(* IEC 61131-3 sources: Word/plc-course/07-timers/labs/starter, 5 files *)

(* ---- 07-1-star-delta.st ---- *)
(* Lab 07-1: Star-delta starter.
   Module 07 (Timers). STARTER - the declarations are done for you;
   write the logic where it says TODO, then run:
     python3 tools/plctest.py 07-timers/labs/starter/07-1-star-delta.st *)

PROGRAM StarDelta
  VAR (* I/O *)
    StartPB       AT %IX0.0 : BOOL;  (* Start push-button, NO: TRUE while pressed *)
    StopPB_NC     AT %IX0.1 : BOOL;  (* Stop push-button, NC: TRUE while NOT pressed *)
    OverloadOK_NC AT %IX0.2 : BOOL;  (* Overload relay contact, NC: TRUE while healthy *)
    MainK         AT %QX0.0 : BOOL;  (* Main (line) contactor *)
    StarK         AT %QX0.1 : BOOL;  (* Star contactor *)
    DeltaK        AT %QX0.2 : BOOL;  (* Delta contactor *)
  END_VAR
  VAR (* settings, e.g. written from an HMI *)
    StarTime : TIME := T#5s;         (* how long the motor starts in star *)
  END_VAR
  VAR (* internal - you may add more variables here *)
    StarTimer : TON;                 (* times the star period *)
    GapTimer  : TON;                 (* changeover dead time, star off -> delta on *)
  END_VAR

  (* TODO: replace these placeholder lines with your logic.
     1. Run latch for MainK (Start, Stop, overload).
     2. StarTimer: star period of StarTime.
     3. GapTimer: 100 ms with both star and delta off.
     4. DeltaK after the gap. Call each timer once per scan, unconditionally. *)
  MainK := FALSE;
  StarK := FALSE;
  DeltaK := FALSE;
END_PROGRAM

CONFIGURATION Config0
  RESOURCE Res0 ON PLC
    TASK MainTask(INTERVAL := T#10ms, PRIORITY := 0);
    PROGRAM Inst0 WITH MainTask : StarDelta;
  END_RESOURCE
END_CONFIGURATION

(* ---- 07-2-flasher-beacon.st ---- *)
(* Lab 07-2: Flasher beacon with separate on and off times.
   Module 07 (Timers). STARTER - the declarations are done for you;
   write the logic where it says TODO, then run:
     python3 tools/plctest.py 07-timers/labs/starter/07-2-flasher-beacon.st *)

PROGRAM FlasherBeacon
  VAR (* I/O *)
    Enable AT %IX0.0 : BOOL;   (* flash request, e.g. "machine about to start" *)
    Beacon AT %QX0.0 : BOOL;   (* beacon lamp *)
  END_VAR
  VAR (* settings, e.g. written from an HMI *)
    OnTime  : TIME := T#500ms; (* lamp on time *)
    OffTime : TIME := T#1s;    (* lamp off time *)
  END_VAR
  VAR (* internal - you may add more variables here *)
    OnTimer  : TON;            (* ON phase *)
    OffTimer : TON;            (* OFF phase *)
  END_VAR

  (* TODO: make Beacon flash: ON for OnTime, OFF for OffTime, repeating while
     Enable is TRUE, always starting with the ON phase. Replace this line. *)
  Beacon := FALSE;
END_PROGRAM

CONFIGURATION Config0
  RESOURCE Res0 ON PLC
    TASK MainTask(INTERVAL := T#10ms, PRIORITY := 0);
    PROGRAM Inst0 WITH MainTask : FlasherBeacon;
  END_RESOURCE
END_CONFIGURATION

(* ---- 07-3-feedback-timeout.st ---- *)
(* Lab 07-3: Motor with run-feedback monitoring.
   Module 07 (Timers). STARTER - the declarations are done for you;
   write the logic where it says TODO, then run:
     python3 tools/plctest.py 07-timers/labs/starter/07-3-feedback-timeout.st *)

PROGRAM FeedbackTimeout
  VAR (* I/O *)
    RunCmd    AT %IX0.0 : BOOL;  (* run request (maintained), TRUE = run *)
    RunFbk    AT %IX0.1 : BOOL;  (* running feedback: contactor aux contact or drive "running" *)
    ResetPB   AT %IX0.2 : BOOL;  (* fault reset push-button, NO *)
    MotorRun  AT %QX0.0 : BOOL;  (* contactor coil / drive run command *)
    FaultLamp AT %QX0.1 : BOOL;  (* fault lamp: on while any fault is latched *)
  END_VAR
  VAR (* settings *)
    StartTimeout : TIME := T#3s;     (* time allowed for feedback after a start *)
    LossDelay    : TIME := T#500ms;  (* feedback dropout tolerated while running *)
  END_VAR
  VAR (* alarms for the HMI *)
    FailToStart : BOOL;          (* latched: no feedback after starting *)
    FbkLost     : BOOL;          (* latched: feedback lost while running *)
  END_VAR
  VAR (* internal - add your own timers and helper variables here *)
    StartTimer : TON;            (* supervises the start *)
    LossTimer  : TON;            (* supervises the running motor *)
  END_VAR

  (* TODO: replace these placeholder lines with your logic.
     - MotorRun follows RunCmd unless a fault is latched.
     - FailToStart: no RunFbk within StartTimeout after a start.
     - FbkLost: RunFbk seen, then missing for LossDelay while running.
     - ResetPB clears the faults only while RunCmd is FALSE. *)
  FailToStart := FALSE;
  FbkLost := FALSE;
  FaultLamp := FALSE;
  MotorRun := FALSE;
END_PROGRAM

CONFIGURATION Config0
  RESOURCE Res0 ON PLC
    TASK MainTask(INTERVAL := T#10ms, PRIORITY := 0);
    PROGRAM Inst0 WITH MainTask : FeedbackTimeout;
  END_RESOURCE
END_CONFIGURATION

(* ---- 07-4-run-hours.st ---- *)
(* Lab 07-4: Accumulating run-hours meter.
   Module 07 (Timers). STARTER - the interface is declared for you;
   add your own internal variables and write the logic where it says TODO,
   then run:
     python3 tools/plctest.py 07-timers/labs/starter/07-4-run-hours.st

   TIME values can be added, subtracted and compared as usual
   (Elapsed := Elapsed + Step; IF Elapsed >= T#1s THEN ...). *)

PROGRAM RunHours
  VAR (* I/O *)
    Running    AT %IX0.0 : BOOL;  (* motor running feedback *)
    ResetPB    AT %IX0.1 : BOOL;  (* reset the meter, e.g. after an overhaul (NO) *)
    ServiceDue AT %QX0.0 : BOOL;  (* service-due lamp *)
  END_VAR
  VAR RETAIN (* on a real PLC the total must survive a power cut *)
    TotalSeconds : DINT;          (* total running time, whole seconds *)
  END_VAR
  VAR (* display values *)
    Hours   : DINT;               (* whole hours *)
    Minutes : DINT;               (* minutes past the whole hour, 0..59 *)
  END_VAR
  VAR (* settings *)
    ServiceHours : DINT := 1000;  (* service interval in running hours *)
  END_VAR
  (* TODO: add a VAR ... END_VAR block here for your timers and helper
     variables (MATIEC does not accept an empty VAR block, so none is given). *)

  (* TODO: replace these placeholder lines with your logic. *)
  TotalSeconds := 0;
  Hours := 0;
  Minutes := 0;
  ServiceDue := FALSE;
END_PROGRAM

CONFIGURATION Config0
  RESOURCE Res0 ON PLC
    TASK MainTask(INTERVAL := T#10ms, PRIORITY := 0);
    PROGRAM Inst0 WITH MainTask : RunHours;
  END_RESOURCE
END_CONFIGURATION

(* ---- 07-5-two-hand-control.st ---- *)
(* Lab 07-5: Two-hand control timing.
   Module 07 (Timers). STARTER - the interface is declared for you;
   write the logic where it says TODO, then run:
     python3 tools/plctest.py 07-timers/labs/starter/07-5-two-hand-control.st

   TRAINING EXERCISE ONLY. Real two-hand control needs safety-rated devices
   and a safety relay or safety PLC (Module 20). *)

PROGRAM TwoHandControl
  VAR (* I/O *)
    LeftPB    AT %IX0.0 : BOOL;  (* left palm button, NO: TRUE while pressed *)
    RightPB   AT %IX0.1 : BOOL;  (* right palm button, NO: TRUE while pressed *)
    PressDown AT %QX0.0 : BOOL;  (* press stroke valve *)
  END_VAR
  VAR (* internal - add your own timers and helper variables here *)
    Window : TON;                (* suggested: time since the first button was pressed *)
  END_VAR

  (* TODO: replace this placeholder line with your logic. *)
  PressDown := FALSE;
END_PROGRAM

CONFIGURATION Config0
  RESOURCE Res0 ON PLC
    TASK MainTask(INTERVAL := T#10ms, PRIORITY := 0);
    PROGRAM Inst0 WITH MainTask : TwoHandControl;
  END_RESOURCE
END_CONFIGURATION
